PROGRAM ctrl_SFC
VAR
END_VAR

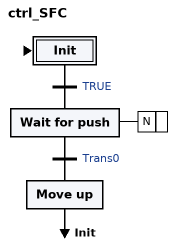
INITIAL_STEP Init:
END_STEP
TRANSITION FROM Init TO Wait_for_push
    := TRUE;
END_TRANSITION
STEP Wait_for_push:  // name as stored: Wait for push
    // ???(N);
END_STEP
TRANSITION FROM Wait_for_push TO Move_up
    := Trans0;
END_TRANSITION
STEP Move_up:  // name as stored: Move up
END_STEP
// no transition between Move up and Init

ACTION act1:

END_ACTION

END_PROGRAM

(* stored: Version 1.1.0.1, ProductVersion 3.1.4022.12
   POU ctrl_SFC: Id {b92edbc5-b47b-48a2-9792-67cc5b3bd0c3}, SpecialFunc None
   Action act1: Id {c4459c8e-8b88-4e27-8541-63b5ec1fc1a2} *)
